RoboDK station: RBT23IT066.rdk

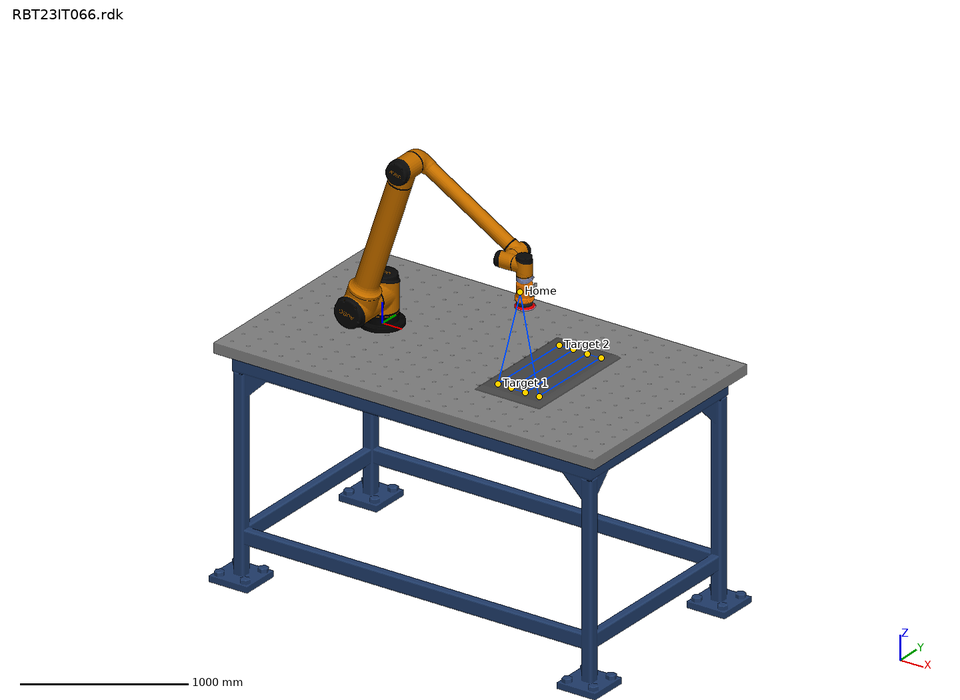
[picture v0: the station drawn from its stored meshes, robots at their saved joint values, targets as dots, program paths as lines]
Station RBT23IT066 (saved by RoboDK 5.9.2). Poses are relative to the parent item; angles as X-Y-Z fixed-axis rotations.
  - frame AUBO-iS20L Base at (0, 0, 0) mm
    - robot AUBO-iS20L: 6 axes
        modified DH rows (alpha deg, a mm, theta deg, d mm): 0, 0, 0, 210.5; 90, 0, 90, 0; 0, 1050, 0, 0; 0, 825, -90, 208; -90, 0, 0, 125; 90, 0, 0, 108.3
        joint limits [-360, -360, -360, -360, -360, -360] to [360, 360, 360, 360, 360, 360]; home [0, -15, 100, 25, 90, 0]; saved at [1.278, -17.993, 103.663, 31.656, 90, 1.278]
      - tool ATI AOV-10 Sander, TCP at (0, 0, 158) mm, size 154.3 x 159.9 x 160.4 mm
    - target Target 1 (Cartesian target) at (1065, -325, 27) mm, rotated rx -180 ry 0 rz 90 deg; joints [152.264, 44.376, 260.344, 125.968, 90, 152.264] of AUBO-iS20L
    - target Target 2 (Cartesian target) at (1065, 315, 27) mm, rotated rx -180 ry 0 rz 90 deg; joints [185.683, 44.281, 260.105, 125.824, 90, 185.683] of AUBO-iS20L
    - target Target 3 (Cartesian target) at (1165, 315, 27) mm, rotated rx -180 ry 0 rz 90 deg; joints [185.206, 47.605, 268.337, 130.733, 90, 185.206] of AUBO-iS20L
    - target Target 4 (Cartesian target) at (1165, -325, 27) mm, rotated rx -180 ry 0 rz 90 deg; joints [154.51, 47.701, 268.571, 130.871, 90, 154.51] of AUBO-iS20L
    - target Target 5 (Cartesian target) at (1265, -325, 27) mm, rotated rx -180 ry 0 rz 90 deg; joints [156.428, 51.383, 277.439, 136.056, 90, 156.428] of AUBO-iS20L
    - target Target 6 (Cartesian target) at (1265, 315, 27) mm, rotated rx -180 ry 0 rz 90 deg; joints [184.802, 51.285, 277.204, 135.92, 90, 184.802] of AUBO-iS20L
    - target Target 7 (Cartesian target) at (1365, 315, 27) mm, rotated rx 180 ry 0 rz 90 deg; joints [184.456, 55.413, 286.943, 141.53, 90, 184.456] of AUBO-iS20L
    - target Target 8 (Cartesian target) at (1365, -325, 27) mm, rotated rx -180 ry 0 rz 90 deg; joints [158.083, 55.516, 287.184, 141.668, 90, 158.083] of AUBO-iS20L
    - target Home (Cartesian target) at (1144.46, -208, 609.76) mm, rotated rx 180 ry 0 rz 90 deg; joints [0, -15, 100, 25, 90, 0] of AUBO-iS20L
  - object Table 1400x800x800mm at (0, 0, 0) mm, size 2795.6 x 1614.4 x 1575 mm, geometry from Table.sld
  - object Display Panel 24in at (1200, 0, -10) mm, rotated rx 0 ry 90 rz 0 deg, size 74.3 x 961.5 x 591.3 mm, geometry from Display-Panel-24in.sld
  - program Prog1 (1 instructions, listed below)
  - program Prog2 (12 instructions, listed below)
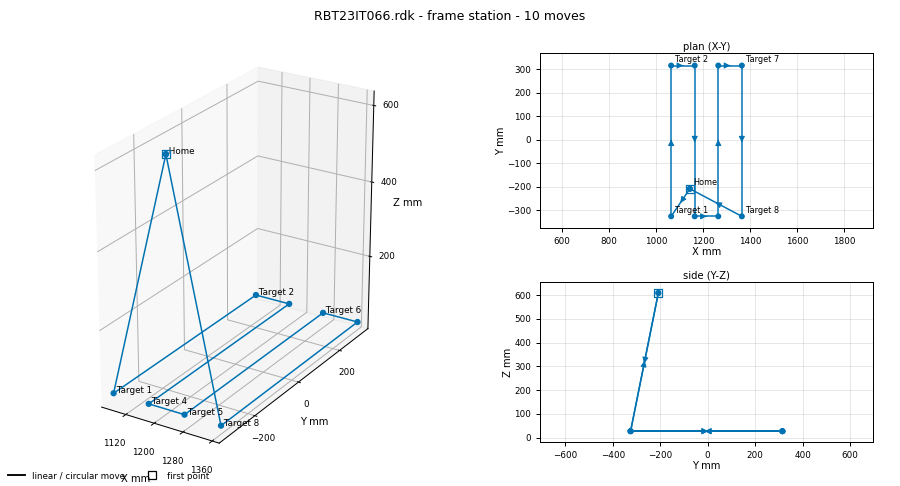
[picture p0: tool path of RBT23IT066.rdk in frame station, 10 of 10 moves have a stored position in this frame; points joined in program order, loops and branches not executed]

--- program Prog1 (robot AUBO-iS20L) ---
  Replace objects

--- program Prog2 (robot AUBO-iS20L) ---
  Set Ref.: AUBO-iS20L Base
  Set Tool: ATI AOV-10 Sander
  MoveL (Home)
  MoveL (Target 1)
  MoveL (Target 2)
  MoveL (Target 3)
  MoveL (Target 4)
  MoveL (Target 5)
  MoveL (Target 6)
  MoveL (Target 7)
  MoveL (Target 8)
  MoveL (Home)
